FUNCTION_BLOCK Q_EndPoint (* Command change end point ( Part 6 - F.26 ) *)
  (* Standard: ISO 11783-6; Description: Copyright (c) 2022 franz This program and the accompanying materials are made available under the terms of the Eclipse Public License 2.0 which is available at https://www.eclipse.org/legal/epl-2.0/ SPDX-License-Identifier: EPL-2.0 see Description Tab *)
  (* Version 1.0, 2022-07-08, franz *)
  (* Documentation:
  Command change end point ( Part 6 - F.26 )
   This command is used to change the end point of a line object by changing the width, height and/or line direction attributes.
   param[in] {objectID, uint16_t}
   Object ID
   param[in] {width_px, uint16_t}
   X value of end point
   param[in] {height_px, uint16_t}
   Y value of end point
   param[in] {direction, uint8_t}
   Line direction
   Return Values: 
   int16_t
    - VT_E_NO_ERR (0) - OK
   - VT_E_OVERFLOW (-6) - buffer overflow
   - VT_E_NOACT (-8) - Command not possible in current state
   - VT_E_NO_INSTANCE (-21) - No VT client available
   - VT_E_ISO_INSTANCE_INVALID (-129) - Identifier for instance (connection) invalid
   - VT_E_NOT_ALIVE (-130) - Identifier for instance valid, but VT Dead.
  *)
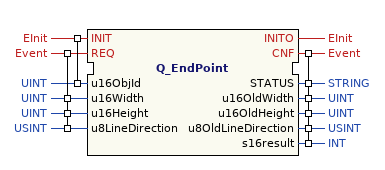
  EVENT_INPUT
    INIT : EInit WITH u16ObjId; (* Service Initialization *)
    REQ WITH u16Width, u16Height, u8LineDirection; (* Service Request *)
  END_EVENT
  EVENT_OUTPUT
    INITO : EInit; (* Initialization Confirm *)
    CNF WITH STATUS, u8OldLineDirection, u16OldWidth, u16OldHeight, s16result; (* Confirmation of Requested Service *)
  END_EVENT
  VAR_INPUT
    u16ObjId : UINT; (* Object ID *)
    u16Width : UINT; (* X value of end point *)
    u16Height : UINT; (* Y value of end point *)
    u8LineDirection : USINT; (* Line direction see Part 6 - B.27 *)
  END_VAR
  VAR_OUTPUT
    STATUS : STRING; (* Service Status *)
    u16OldWidth : UINT; (* Old X value of end point *)
    u16OldHeight : UINT; (* Old Y value of end point *)
    u8OldLineDirection : USINT; (* Old line direction see Part 6 - B.27 *)
    s16result : INT; (* retval see description *)
  END_VAR
END_FUNCTION_BLOCK
